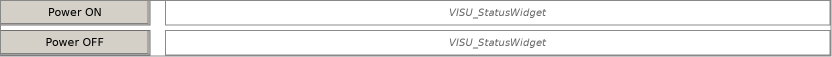
VISUALIZATION VISU_Axes_Commands_Power  // 832x57
VAR_IN_OUT
	powerOn : AxesPowerOnProcess;
    powerOff : AxesPowerOffProcess;
    
    powerOnStatus : StatusWidget;
    powerOffStatus : StatusWidget;
    
END_VAR
    Button (0,0 150x25), "Power ON", input disabled if: powerOn.statuses.enabledStatus.disabled
        OnMouseClick: execute { powerOn.request(); }
    Button (0,30 150x25), "Power OFF", input disabled if: powerOff.statuses.enabledStatus.disabled
        OnMouseClick: execute { powerOff.request(); }
    Frame (165,0 665x25)
        shows VISU_StatusWidget(widget := powerOnStatus)
    Frame (165,30 665x25)
        shows VISU_StatusWidget(widget := powerOffStatus)
END_VISUALIZATION

(* stored: Version 1.1.0.1, ProductVersion 3.1.4019.2
   Visu VISU_Axes_Commands_Power: Id {9c819088-2be7-45c5-977d-87d8155e463a} *)
